(* CODESYS project FU_sConcat6.xml

Project tree, tasks and I/O mapping:
  function FU_sConcat6 [ST]
*)

// FU_sConcat6
//This functions combines six strings
// |**Version**|**Author**| **Date** |**Changes**
// | 1         | NSN      | 03-12-18 | Creation
FUNCTION FU_sConcat6 : STRING(255)
VAR_INPUT
	s1			:STRING(255);			//Input String1
	s2			:STRING(255);			//Input String2
	s3			:STRING(255);			//Input String3
	s4			:STRING(255);			//Input String4
	s5			:STRING(255);			//Input String5
	s6			:STRING(255);			//Input String6
END_VAR

FU_sConcat6BIBO(sOut:=ADR(FU_sConcat6),s1:=ADR(s1),s2:=ADR(s2),s3:=ADR(s3),s4:=ADR(s4),s5:=ADR(s5),s6:=ADR(s6),wOutSize:=255);

END_FUNCTION
